# EPICS autosave request: iocBoot/iocrsfsl/auto_settings_RSFSL.req
file "RSFSL_settings.req",                P=$(P),  R=$(R)
